PROGRAM prgComEffIO
VAR
	fbCom		: FB_MqttCommunicator_V2;
	int_PowerLinkNumber: INT;
END_VAR

fbCom(
	bConnect:= TRUE, 
	strAuthkey := 'EIO08031879806',
	sUserName:= , 			// see below
	sUserPassword:= , 		// see below
	eSavePositionCertificate:= eSavePositionOnPLC.ePostionHardDisk, 
	bConnected=> , 
	bError=> , 
	hrErrorCode=> , 
	eConnectionState=> , 
	eErrorMessage_Out=> );



prg_ReadDeviceName();
IF prg_ReadDeviceName.sDeviceName = '' THEN
	prg_ReadDeviceName.bStart := TRUE;
END_IF

// select user / pass according device name:
 IF prg_ReadDeviceName.sDeviceName = 'EIOSP000001' THEN   // powerlink #1
	fbCom.sUserName:= '8db75f2f-db57-48ff-b140-11662b7a588b'; 
	fbCom.sUserPassword:= '39361e12-8154-402f-92ce-60848a86714e';
	prgEM.uiCurrentTransformerRatio_EM1	:= 300;
	prgEM.uiCurrentTransformerRatio_EM2	:= 32;
	prgEM.uiCurrentTransformerRatio_EM3	:= 32;
	prgEM.uiCurrentTransformerRatio_EM4	:= 32;
	prgEM.uiCurrentTransformerRatio_EM5	:= 32;
	prgEM.uiCurrentTransformerRatio_EM6	:= 32;
	prgEM.uiCurrentTransformerRatio_EM7	:= 32;
	

END_IF

END_PROGRAM

(* stored: Version 1.1.0.1, ProductVersion 3.1.4024.12
   POU prgComEffIO: Id {cbcd318b-bf51-484c-bcaa-d6efcdf43fe3}, SpecialFunc None *)
